(* CODESYS project CowbellCheckers_Tracy.project

Project tree, tasks and I/O mapping:
  Device : PAC320-CXX2X-XX, Parker Hannifin, order no. PAC320-CXX2X-XX, version 3.5.9.10
    application Application
      task EtherCAT_Master (externalevent, external event EVENT_ECM_DC, priority 0) calls EtherCAT_Master.EtherCAT_Task [EtherCAT_Master.EtherCAT_Task], MainProgram
      task VISU_TASK (cyclic, interval 100 ms, priority 31) calls VisuElems.Visu_Prg
      SymbolConfiguration
    SoftMotion General Axis Pool
    EtherCAT_Master : PAC320 EtherCAT Master, Parker Hannifin, order no. PAC320-XXXXX-XX, version 3.5.9.10
      PAC320_BusCoupler : PAC320 BusCoupler, Parker Hannifin, version Revision=16#00000001
          settings: StationAlias = 0; DC sync0 cycletime = 4000; DC sync1 cycletime = 4000
        PACIO_DI16_DO16 : DI16/DO16 1ms 0.5A (PACIO-450-03), Parker Hannifin, version Revision=16#00000001
            settings: StationAlias = 0; DC sync0 cycletime = 4000; DC sync1 cycletime = 4000
            unmapped channels: DigitalOutput0, DigitalOutput1, DigitalOutput2, DigitalOutput3, DigitalOutput4, DigitalOutput5, DigitalOutput6, DigitalOutput7, DigitalOutput8, DigitalOutput9, DigitalOutput10, DigitalOutput11, DigitalOutput12, DigitalOutput13, DigitalOutput14, DigitalOutput15, DigitalInput0, DigitalInput1, DigitalInput2, DigitalInput3, DigitalInput4, DigitalInput5, DigitalInput6, DigitalInput7, DigitalInput8, DigitalInput9, DigitalInput10, DigitalInput11, DigitalInput12, DigitalInput13, DigitalInput14, DigitalInput15
      PD_xxC_Standard_EtherCAT_drive : PD-xxC - Standard EtherCAT drive(CoE,EoE,FoE) V2.0, Parker Hannifin, version Revision=16#00000002
          settings: DC sync0 cycletime = 4000
          unmapped channels: Controlword, Target Position, Touch Probe Function, Digital Ouputs, Statusword, Position Actual Value, Following Error Actual Value, Touch Probe Status, Touch Probe 1 Positive Edge Position Value, Digital Inputs
        X : SM_Drive_GenericDSP402, 3S - Smart Software Solutions GmbH, order no. 0, version 4.0.0.0
            settings: wDriveID = 3; AdrOffset_8010 = 4; BitOffset_8010 = 0; BitLength_8010 = 16; Address_8010 = '%QW2'; Type_8010 = 'UINT'; AddressPointer_8010 = ADR(%QW2); AdrOffset_8020 = 8; BitOffset_8020 = 0; BitLength_8020 = 32; Address_8020 = '%QD2'; Type_8020 = 'DINT'; AddressPointer_8020 = ADR(%QD2); AdrOffset_8030 = 4294967295; BitOffset_8030 = 0; BitLength_8030 = 0; Address_8030 = ''; Type_8030 = ''; AddressPointer_8030 = 0; AdrOffset_8040 = 4294967295; BitOffset_8040 = 0; BitLength_8040 = 0; Address_8040 = ''; Type_8040 = ''; AddressPointer_8040 = 0; AdrOffset_8050 = 4294967295; BitOffset_8050 = 0; BitLength_8050 = 0; Address_8050 = ''; Type_8050 = ''; AddressPointer_8050 = 0; AdrOffset_8060 = 12; BitOffset_8060 = 0; BitLength_8060 = 16; Address_8060 = '%QW6'; Type_8060 = 'UINT'; AddressPointer_8060 = ADR(%QW6); AdrOffset_8070 = 4294967295; BitOffset_8070 = 0; BitLength_8070 = 0;
              Address_8070 = ''; Type_8070 = ''; AddressPointer_8070 = 0; AdrOffset_8080 = 4294967295; BitOffset_8080 = 0; BitLength_8080 = 0; Address_8080 = ''; Type_8080 = ''; AddressPointer_8080 = 0; AdrOffset_8090 = 16; BitOffset_8090 = 0; BitLength_8090 = 32; Address_8090 = '%QD4'; Type_8090 = 'UDINT'; AddressPointer_8090 = ADR(%QD4); AdrOffset_8510 = 4; BitOffset_8510 = 0; BitLength_8510 = 16; Address_8510 = '%IW2'; Type_8510 = 'UINT'; AddressPointer_8510 = ADR(%IW2); AdrOffset_8520 = 8; BitOffset_8520 = 0; BitLength_8520 = 32; Address_8520 = '%ID2'; Type_8520 = 'DINT'; AddressPointer_8520 = ADR(%ID2); AdrOffset_8530 = 4294967295; BitOffset_8530 = 0; BitLength_8530 = 0; Address_8530 = ''; Type_8530 = ''; AddressPointer_8530 = 0; AdrOffset_8540 = 4294967295; BitOffset_8540 = 0; BitLength_8540 = 0; Address_8540 = ''; Type_8540 = ''; AddressPointer_8540 = 0; AdrOffset_8550 = 4294967295;
              BitOffset_8550 = 0; BitLength_8550 = 0; Address_8550 = ''; Type_8550 = ''; AddressPointer_8550 = 0; AdrOffset_8560 = 24; BitOffset_8560 = 0; BitLength_8560 = 32; Address_8560 = '%ID6'; Type_8560 = 'UDINT'; AddressPointer_8560 = ADR(%ID6); AdrOffset_8570 = 16; BitOffset_8570 = 0; BitLength_8570 = 16; Address_8570 = '%IW8'; Type_8570 = 'UINT'; AddressPointer_8570 = ADR(%IW8); AdrOffset_8580 = 20; BitOffset_8580 = 0; BitLength_8580 = 32; Address_8580 = '%ID5'; Type_8580 = 'DINT'; AddressPointer_8580 = ADR(%ID5); AdrOffset_8590 = 4294967295; BitOffset_8590 = 0; BitLength_8590 = 0; Address_8590 = ''; Type_8590 = ''; AddressPointer_8590 = 0; AdrOffset_8600 = 4294967295; BitOffset_8600 = 0; BitLength_8600 = 0; Address_8600 = ''; Type_8600 = ''; AddressPointer_8600 = 0; AdrOffset_8600 = 4294967295; BitOffset_8600 = 0; BitLength_8600 = 0; Address_8610 = ''; Type_8610 = '';
              AddressPointer_8610 = 0; AdrOffset_8620 = 12; BitOffset_8620 = 0; BitLength_8620 = 32; Address_8620 = '%ID3'; Type_8620 = 'DINT'; AddressPointer_8620 = ADR(%ID3)
  CODESYS_SoftMotion_Win_V3 : CODESYS SoftMotion Win V3, 3S - Smart Software Solutions GmbH, order no. 309021, version 3.5.9.10
    application Application
      libraries: PAC Help Library, 0.1 (Parker ); SysFile, 3.5.9.0 (System); CmpErrors, 3.3.1.40 (System); ISysTypes2, 3.5.0.0 (System); SysTimeRtc, 3.5.5.0 (System); SysTimeCore, 3.5.5.0 (System); Util, 3.5.9.0 (System)
      task Main (cyclic, interval 4000 ms, priority 0) calls TestInitialization, TestMyArray
      task VISU_TASK (cyclic, interval 100 ms, priority 31) calls VisuElems.Visu_Prg
      SymbolConfiguration
      Visualizations/
        visualisation Enable
        visualisation OnePlayer
        visualisation InitScreen
        visualisation MainView
        visualisation GameView
        visualisation HowToPlay
        visualisation History
      program TestMyArray [ST]
      global variables PersistentVars
      data type History
      function block ArrayMove [ST]
      program LogData [ST]
      function GetHeaderString [ST]
      function GetTimeStampString [ST]
      program LogWinnerNames [ST]
      function GetLogMsgString [ST]
      visualisation ExportData
    SoftMotion General Axis Pool
      X : SM_Drive_Virtual, 3S - Smart Software Solutions GmbH, order no. 1805, version 4.0.0.0
          settings: wDriveID = 4
      Y : SM_Drive_Virtual, 3S - Smart Software Solutions GmbH, order no. 1805, version 4.0.0.0
          settings: wDriveID = 5
      Z : SM_Drive_Virtual, 3S - Smart Software Solutions GmbH, order no. 1805, version 4.0.0.0
          settings: wDriveID = 6
  text COWBELL_PROGRAMMING_STANDARD
  global variables GlobalVars
  text list GlobalTextList
  function block Initialization [CFC]
  program TestInitialization [CFC]
*)

// CODESYS_SoftMotion_Win_V3/Application/History
TYPE History :
STRUCT
	
	Names: STRING;
	Moves: INT;
	
END_STRUCT
END_TYPE

// GlobalVars
(* COWBELL GLOBAL VARIABLES *)
VAR_GLOBAL
	systemEnable : BOOL;
	
	
	p1CheckerColor: DWORD := 16#FFFFFFFF; // 16# - interpret as hexidecimal, FF - transparency (Fully Opaque, 00 fully transparent), FF - Red, FF - Green, FF - Blue
	p2CheckerColor: DWORD := 16#FF000000;
	
	p1DefaultName: STRING := 'Player_1';
	p2DefaultName: STRING := 'Player_2';
	
	winnerName: STRING := 'Default';
	winnerMoves: INT := 4;
	
	//Export data global variables
	
	g_PosDistance:REAL := 20.0;
	g_NegDistance:REAL := -20.0;
	g_Vel:REAL := 5.0;
	g_Acc:REAL := 10.0;
	//In_Power : BOOL ;
	//In_Reset : BOOL;
	//In_Pos : BOOL;
	//In_Neg : BOOL;
	//In_Stop : BOOL;
	//In_Zero : BOOL;
	g_MoveDwellPos : BOOL := FALSE;
	g_MoveDwellNeg : BOOL := FALSE;
	g_MoveDwellPos_Y : BOOL := FALSE;
	g_MoveDwellNeg_Y : BOOL := FALSE;
	g_MoveDwellPos_Z : BOOL := FALSE;
	g_MoveDwellNeg_Z : BOOL := FALSE;
	g_MoveDwellPos_A : BOOL := FALSE;
	g_MoveDwellNeg_A : BOOL := FALSE;
	g_GotSDO_PostionPos : BOOL;
	g_GotSDO_PostionNeg : BOOL;
	g_GotSDO_Y_PostionPos : BOOL;
	g_GotSDO_Y_PostionNeg : BOOL;
	DC_InSync: BOOL;
	g_FirstSync: BOOL;
	g_LostSync: BOOL;
	
	
	//ScanTimeMax: DINT;
	//ScanTimeMin: DINT;
	//dcWindow: WORD := 50;

	//MaxScanTime: DINT;
	//MaxSyncTime: DINT;
	//MinSyncTime: DINT;
	//MaxTotalSyncBufferAvg: DINT;
	MyArray: ARRAY[0..9, 0..9] OF REAL;
	
END_VAR

// CODESYS_SoftMotion_Win_V3/Application/PersistentVars
{attribute 'qualified_only'}
VAR_GLOBAL PERSISTENT RETAIN
	MyArray : ARRAY [1..20] OF History;
END_VAR

// TestInitialization
PROGRAM TestInitialization
VAR
	Initialization_0: Initialization;
	X_enable: BOOL;
	X_reset: BOOL;
	
END_VAR

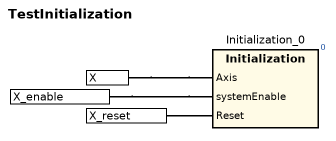
Initialization_0(Axis := X, systemEnable := X_enable, Reset := X_reset); // Initialization

END_PROGRAM

// Initialization
FUNCTION_BLOCK Initialization
VAR_IN_OUT
	Axis: SM3_Basic.AXIS_REF_SM3;
	END_VAR
VAR_INPUT
	systemEnable : BOOL;
	Reset:BOOL;     // reset the drive
	
	
END_VAR
VAR_OUTPUT
END_VAR
VAR
	MC_Power_X: MC_Power;
	MC_Power_Y: MC_Power;
	MC_Power_Z: MC_Power;
	MC_Reset_X: MC_Reset;
	MC_Reset_Y: MC_Reset;
	MC_Reset_Z: MC_Reset;
	MC_Jog_X: MC_Jog;
END_VAR

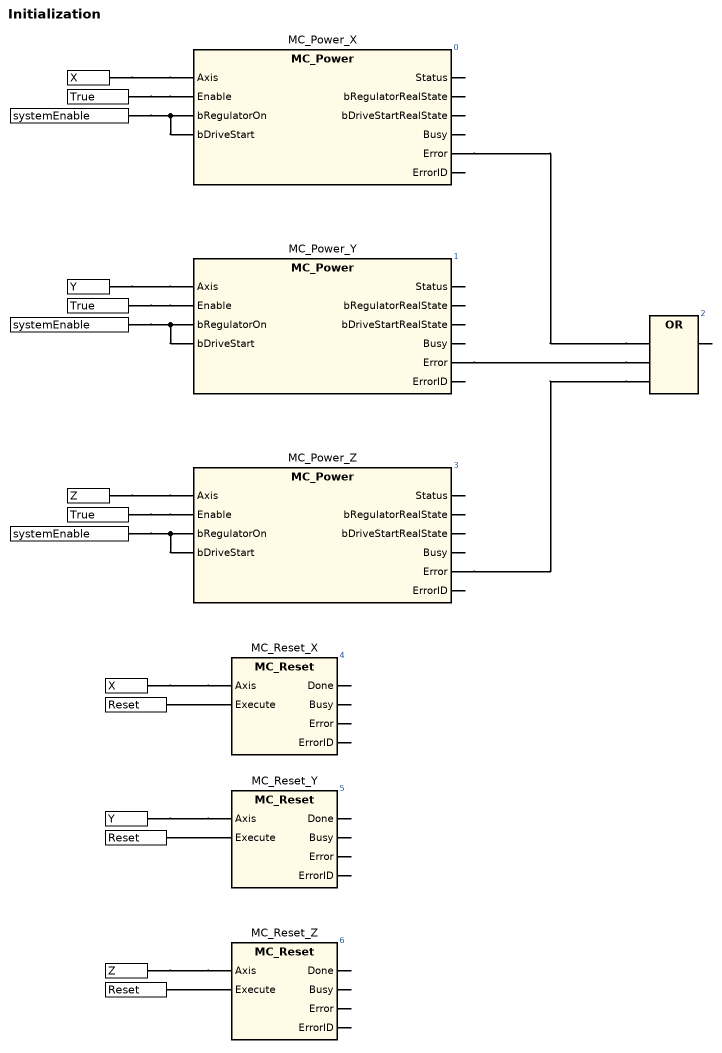
MC_Power_X(Axis := X, Enable := True, bRegulatorOn := systemEnable, bDriveStart := systemEnable); // MC_Power
MC_Power_Y(Axis := Y, Enable := True, bRegulatorOn := systemEnable, bDriveStart := systemEnable); // MC_Power
(* MC_Power_X.Error OR MC_Power_Y.Error OR MC_Power_Z.Error; result not used *)
MC_Power_Z(Axis := Z, Enable := True, bRegulatorOn := systemEnable, bDriveStart := systemEnable); // MC_Power
MC_Reset_X(Axis := X, Execute := Reset); // MC_Reset
MC_Reset_Y(Axis := Y, Execute := Reset); // MC_Reset
MC_Reset_Z(Axis := Z, Execute := Reset); // MC_Reset

END_FUNCTION_BLOCK

// CODESYS_SoftMotion_Win_V3/Application/TestMyArray
PROGRAM TestMyArray
VAR
	k : INT ; 
	arrayTest : ArrayMove;
END_VAR

arrayTest();
//k := ArrayMove.TestArray[2];

END_PROGRAM

// CODESYS_SoftMotion_Win_V3/Application/ArrayMove
FUNCTION_BLOCK ArrayMove
VAR_INPUT
	//TestArray: ARRAY [1..20] OF INT := [1,2,3,4,5,6,7,8,9,10,11,12,13,14,15,16,17,18,19,20];
	i: INT ; 
END_VAR
VAR_OUTPUT
END_VAR
VAR
	Done : BOOL;
END_VAR

IF(NOT Done) THEN
	
FOR i:= 20 TO 2 BY -1 DO 
	PersistentVars.MyArray[i]:= PersistentVars.MyArray [i-1];
END_FOR
PersistentVars.MyArray[1].Names := winnerName;
PersistentVars.MyArray[1].Moves := winnerMoves;
Done := TRUE;
END_IF

END_FUNCTION_BLOCK

// CODESYS_SoftMotion_Win_V3/Application/LogData
PROGRAM LogData
VAR
	filename: STRING := '/Windows/Logs/Log_HighCycleCount.csv';
	filehandle: SYSFILE.RTS_IEC_HANDLE;
	strMsg: STRING[255];
	FOResult: SYSFILE.RTS_IEC_RESULT;
	FWResult: SYSFILE.RTS_IEC_RESULT;
	FWStatus: POINTER TO RTS_IEC_RESULT;
	FCResult: SYSFILE.RTS_IEC_RESULT;
	bytesWritten: DWORD;
	bFileOpen: BOOL;
	iStatus : INT := 0;
	
	
	SafeToStop: BOOL;
	Result1: SYSFILE.RTS_IEC_RESULT;
	SizeFile: DWORD;
	ErrorID: INT;
	diActPosition: UDINT;
	
	LogIndex :DINT := 0;
	LogMsg : ARRAY [1..200] OF STRING[255];
	LogType : STRING;

	intIndex: DINT;
	

END_VAR

CASE iStatus OF
	1: //Open File
	
	SafeToStop := FALSE;
	filehandle := SysFileOpen(szFile := filename, am := sysfile.AM_WRITE, pResult:= ADR(FOResult));
	IF (filehandle <> 16#00000000 AND filehandle <> 16#FFFFFFFF AND FOResult = cmperrors.Errors.ERR_OK) THEN 
		bFileOpen := TRUE;
		iStatus := iStatus + 1;
	ELSE
		ErrorID := -1 * iStatus;  //Open Memory Copy Failed
		iStatus := 99;
	END_IF//Open File

2:	//Log Data
	FOR intIndex := 1 TO LogIndex DO
		strMsg := LogMsg[intIndex];
		bytesWritten:= SysFileWrite(filehandle, ADR(strMsg), DINT_TO_DWORD(LEN(strMsg)), ADR(FWResult));
		IF FWResult <> CmpErrors.Errors.ERR_OK THEN
			ErrorID := -1 * iStatus;  //Log Data Failed
			iStatus := 100;
		END_IF
	END_FOR

3:  //Close File
	FCResult := SysFileClose(filehandle);
	IF FCResult = CmpErrors.Errors.ERR_OK THEN
		SafeToStop:=TRUE;
		iStatus := 5;
	ELSE
		ErrorID := -1 * iStatus;  //File Close Failed
		iStatus := 99;
	END_IF
END_CASE

END_PROGRAM

// CODESYS_SoftMotion_Win_V3/Application/GetHeaderString
FUNCTION GetHeaderString : STRING[255]
VAR_INPUT
END_VAR
VAR
	msg: STRING[255];
	seperator: STRING;
	eol:String;
	strTemp0 : STRING[255];
	strTemp1 : STRING[255];
	

END_VAR

eol := WORD_AS_STRING(16#0A0D, FALSE);
seperator := ',';

strTemp0 := Concat(Concat(	'Winners', 
						 seperator), 
						    'Moves');




GetHeaderString := Concat(Concat(Concat(Concat(	'TimeStamp', 
														seperator),
														strTemp0), 
														seperator),
						     								eol);

END_FUNCTION

// CODESYS_SoftMotion_Win_V3/Application/GetTimeStampString
FUNCTION GetTimeStampString : STRING
VAR_INPUT
END_VAR
VAR
	TimeStamp : SysTime;
	StructTimeStamp : SysTimeDate;
	Result : RTS_IEC_RESULT;
	StrDate : STRING;
	StrTime : STRING;
	

END_VAR

Result := systimertc.SysTimeRtcHighResGet(pTimestamp := TimeStamp);

Result := systimertc.SysTimeRtcConvertHighResToLocal(pTimeStamp:=TimeStamp, pDate:=StructTimeStamp);

StrDate := UINT_TO_STRING(StructTimeStamp.wYear);
IF StructTimeStamp.wMonth < 10 THEN 
	StrDate := Concat(Concat(StrDate, '0') , UINT_TO_STRING(StructTimeStamp.wMonth));
ELSE
	StrDate := Concat(StrDate , UINT_TO_STRING(StructTimeStamp.wMonth));
END_IF

IF StructTimeStamp.wDay < 10 THEN 
	StrDate := Concat(Concat(StrDate , '0') , UINT_TO_STRING(StructTimeStamp.wDay));
ELSE
	StrDate := Concat(StrDate , UINT_TO_STRING(StructTimeStamp.wDay));
END_IF


IF StructTimeStamp.wHour < 10 THEN 
	StrTime := Concat(Concat('0' , UINT_TO_STRING(StructTimeStamp.wHour)) , ':');
ELSE
	StrTime := Concat(UINT_TO_STRING(StructTimeStamp.wHour) , ':');
END_IF

IF StructTimeStamp.wMinute < 10 THEN 
	StrTime := Concat(Concat(Concat(StrTime , '0') , UINT_TO_STRING(StructTimeStamp.wMinute)), ':');
ELSE
	StrTime := Concat(Concat(StrTime , UINT_TO_STRING(StructTimeStamp.wMinute)), ':');
END_IF

IF StructTimeStamp.wSecond < 10 THEN 
	StrTime := Concat(Concat(Concat(StrTime , '0') , UINT_TO_STRING(StructTimeStamp.wSecond)) , '.');
ELSE
	StrTime := Concat(Concat(StrTime , UINT_TO_STRING(StructTimeStamp.wSecond)) , '.');
END_IF

IF StructTimeStamp.wMilliseconds < 10 THEN 
	StrTime := Concat(Concat(StrTime , '00') , UINT_TO_STRING(StructTimeStamp.wMilliseconds));
ELSE
	IF StructTimeStamp.wMilliseconds < 100 THEN 
		StrTime := Concat(Concat(StrTime , '0') , UINT_TO_STRING(StructTimeStamp.wMilliseconds));
	ELSE
		StrTime := Concat(StrTime , UINT_TO_STRING(StructTimeStamp.wMilliseconds));
	END_IF
END_IF

//GetTimeStampString := Concat(Concat(strDate , '-'), strTime);
GetTimeStampString := strTime;

END_FUNCTION

// CODESYS_SoftMotion_Win_V3/Application/LogWinnerNames
PROGRAM LogWinnerNames
VAR
	strMsg: STRING[255];
	iStatus : INT := 0;
	LogIndex :DINT := 0;
	LogMsg : ARRAY [1..200] OF STRING[255];
	LogType : STRING;
	
	CycleTimeWarning: DWORD := 600;
	TotalSyncBufferAvgWarning: DINT := 125;
	CycleTimeError: DWORD := 900;
	TotalSyncBufferAvgError: DINT := 200;
	
	
	
END_VAR

VAR_INPUT
	bResetArray: BOOL;
END_VAR

IF bResetArray = TRUE THEN
	LogIndex := 0;
END_IF




CASE iStatus OF
	

0:	//Log Data
	LogIndex := LogIndex + 1;
	
	LogMsg[LogIndex] :=  GetLogMsgString();
	
	iStatus := 2;

END_CASE

END_PROGRAM

// CODESYS_SoftMotion_Win_V3/Application/GetLogMsgString
FUNCTION GetLogMsgString : STRING[255]
VAR_INPUT
END_VAR
VAR
	msg: STRING[255];
	seperator: STRING;
	eol:String;
	
	DataPrep: STRING[255];
	
	
END_VAR

eol := WORD_AS_STRING(16#0A0D, FALSE);
seperator := ',';


DataPrep := Concat(Concat(  PersistentVars.MyArray[1].Names,
                                                  seperator),
            INT_TO_STRING(PersistentVars.MyArray[1].Moves));
																												



GetLogMsgString := Concat(Concat(Concat(Concat(	GetTimeStampString(),
														seperator),
														DataPrep), 
														seperator),
															eol);

END_FUNCTION

// CODESYS_SoftMotion_Win_V3/Application/Visualizations/Enable
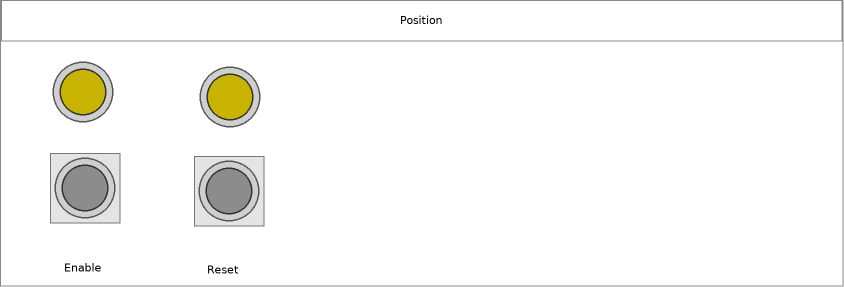
VISUALIZATION Enable  // 844x287
    Frame (1,0 841x41), "Position", text variable: X
        shows SM3_Basic.LinDrive(m_Input_AXISREF := X)
    Label (8,253 150x30), "Enable"
    PushSwitch (50,153 70x70), variable: TestInitialization.X_enable, behaviour: TOGGLE, style: Switch-PushSwitch-Gray
    Lamp1 (48,57 70x70), variable: TestInitialization.X_enable, style: Lamp-Lamp1-Yellow
    PushSwitch (194,156 70x70), variable: TestInitialization.X_reset, behaviour: TOGGLE, style: Switch-PushSwitch-Gray
    Lamp1 (195,62 70x70), variable: TestInitialization.X_reset, style: Lamp-Lamp1-Yellow
    Label (148,255 150x30), "Reset"
END_VISUALIZATION

// CODESYS_SoftMotion_Win_V3/Application/Visualizations/OnePlayer
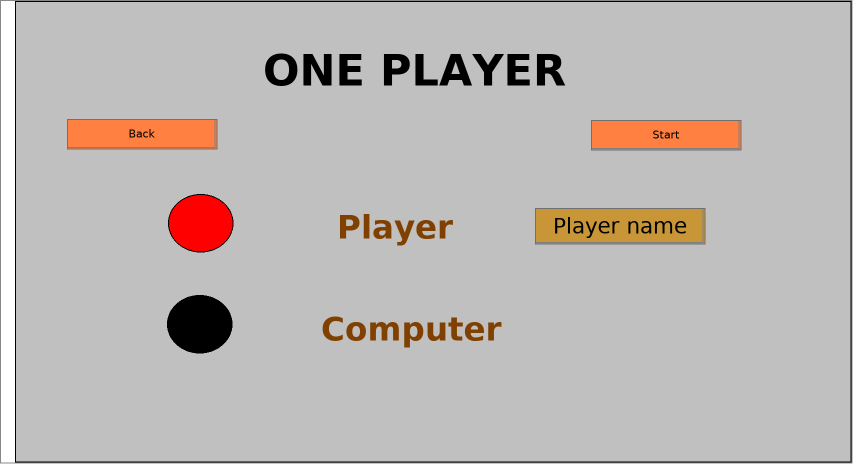
VISUALIZATION OnePlayer  // 853x464
    Rectangle (15,1 836x461)
    Label (230,22 369x97), "ONE PLAYER"
    Button (67,119 150x30), "Back"
    Button (591,120 150x30), "Start"
    Label (326,203 138x48), "Player"
    Button (535,208 170x36), "Player name"
    Ellipse (168,194 65x58)
    Ellipse (167,295 65x58)
    Label (281,305 261x48), "Computer"
END_VISUALIZATION

// CODESYS_SoftMotion_Win_V3/Application/Visualizations/InitScreen
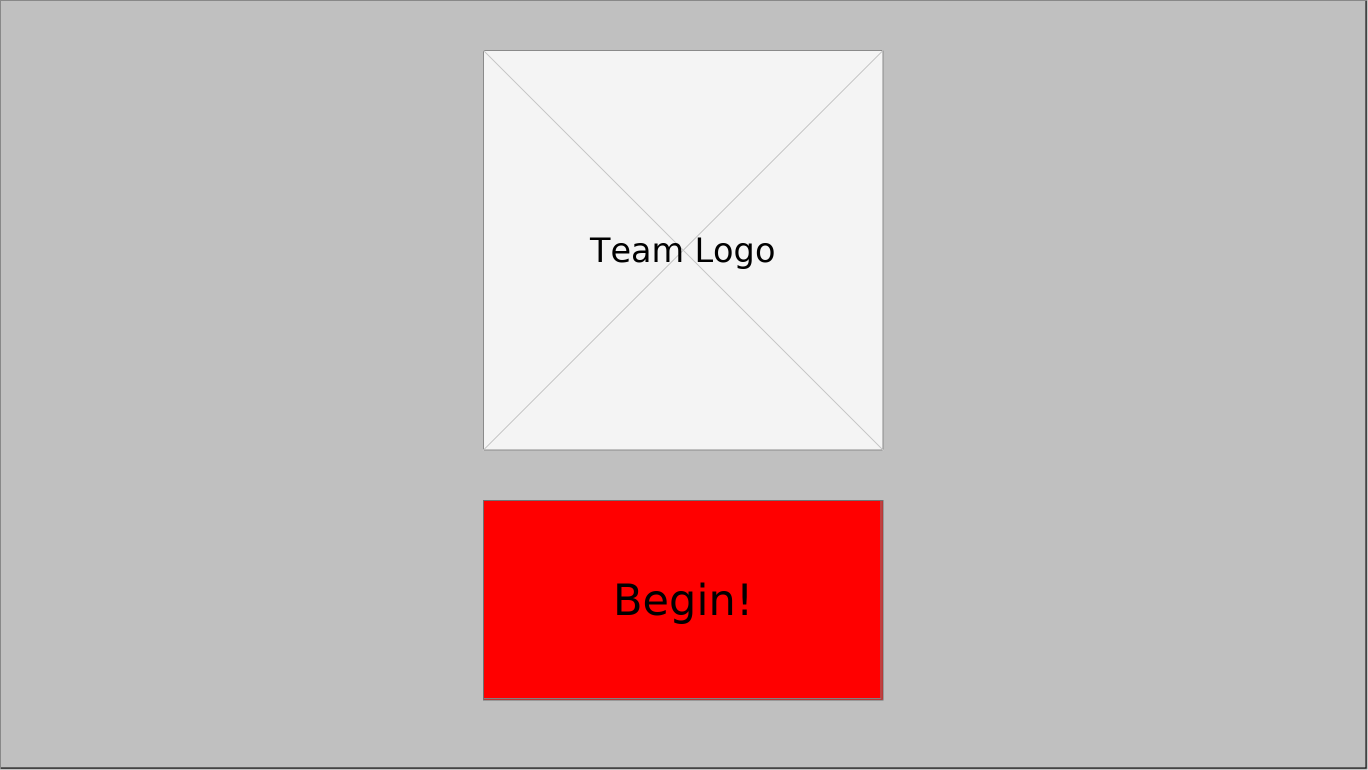
VISUALIZATION InitScreen  // 1368x770
    Rectangle (0,0 1366x768)
    Image (483,50 400x400), "Team Logo"
    Button (483,500 400x200), "Begin!"
END_VISUALIZATION

// CODESYS_SoftMotion_Win_V3/Application/Visualizations/MainView
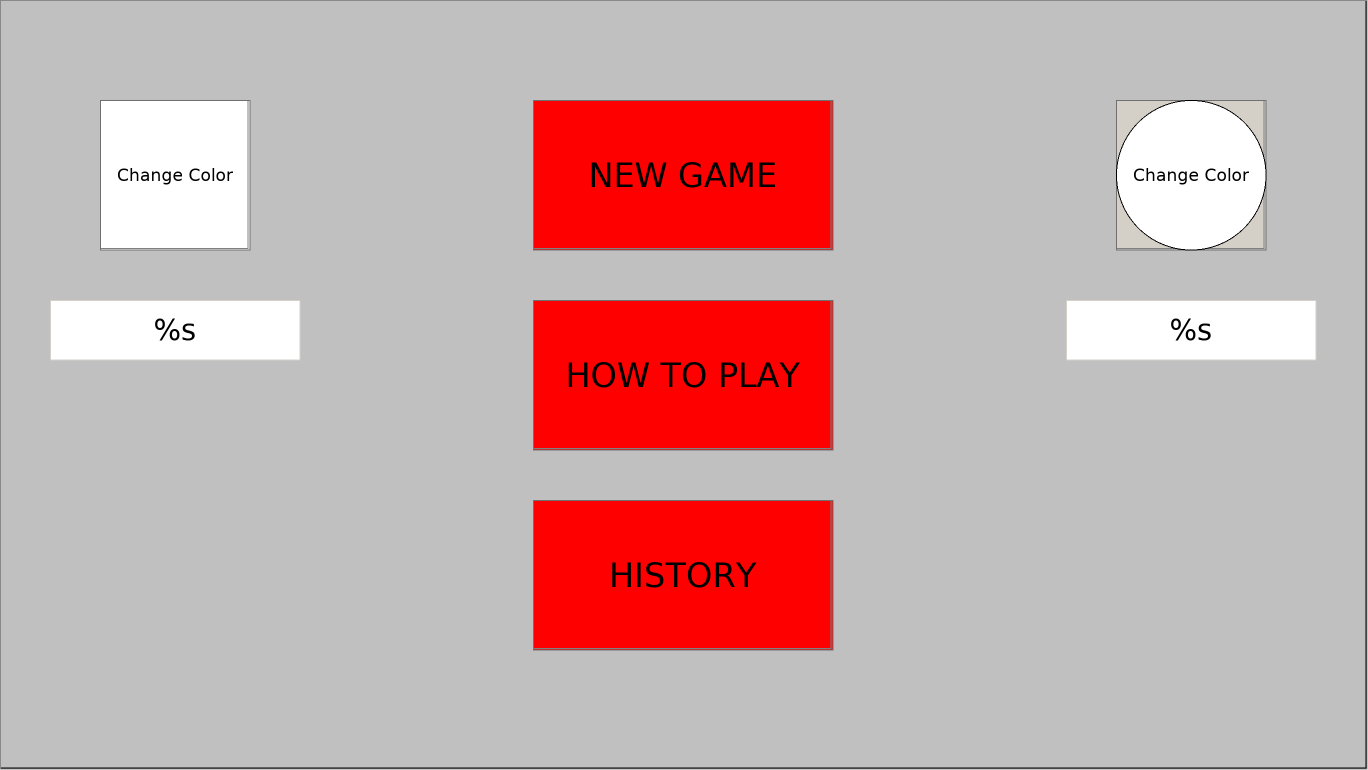
VISUALIZATION MainView  // 1368x770
    Rectangle (0,0 1366x768)
    Ellipse (100,100 150x150), colour variable: p1CheckerColor
    Button (100,100 150x150), "Change Color"
    Button (1116,100 150x150)
    Ellipse (1116,100 150x150), "Change Color", colour variable: p2CheckerColor
    Textfield (50,300 250x60), "%s", text variable: p1DefaultName
    Textfield (1066,300 250x60), "%s", text variable: p2DefaultName
    Button (533,100 300x150), "NEW GAME"
    Button (533,300 300x150), "HOW TO PLAY"
    Button (533,500 300x150), "HISTORY"
END_VISUALIZATION

// CODESYS_SoftMotion_Win_V3/Application/Visualizations/GameView
VISUALIZATION GameView  // 2x2
END_VISUALIZATION

// CODESYS_SoftMotion_Win_V3/Application/Visualizations/HowToPlay
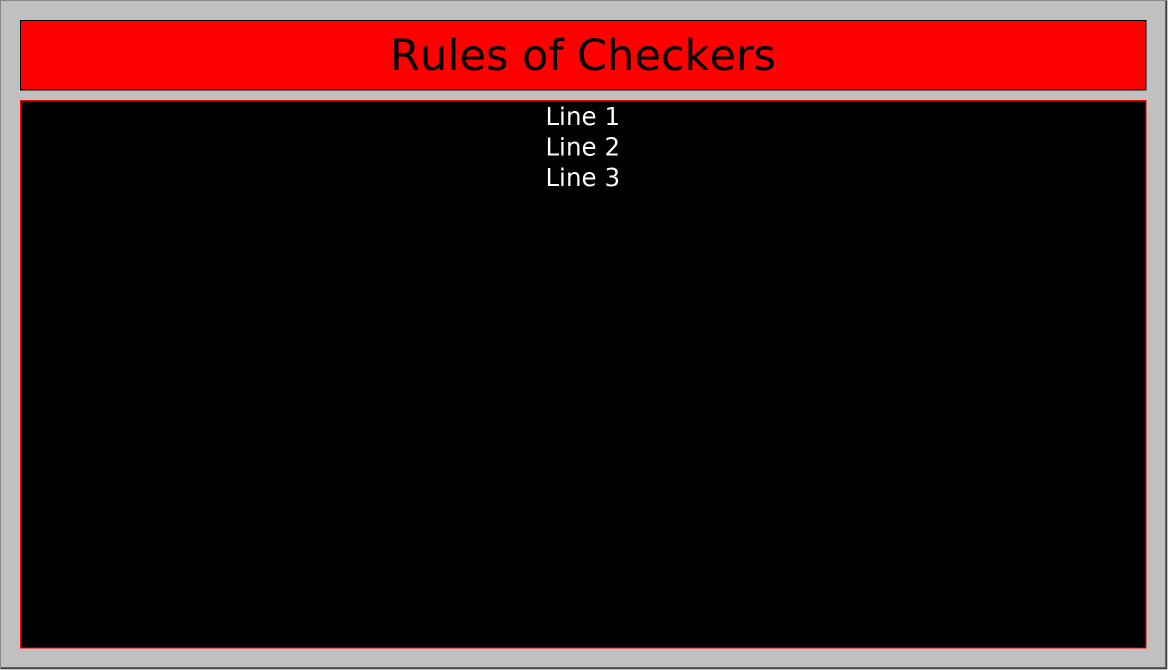
VISUALIZATION HowToPlay  // 1168x670
    Rectangle (0,0 1166x668)
    Textfield (20,100 1126x548), "Line 1 Line 2 Line 3"
    Textfield (20,20 1126x70), "Rules of Checkers"
END_VISUALIZATION

// CODESYS_SoftMotion_Win_V3/Application/Visualizations/History
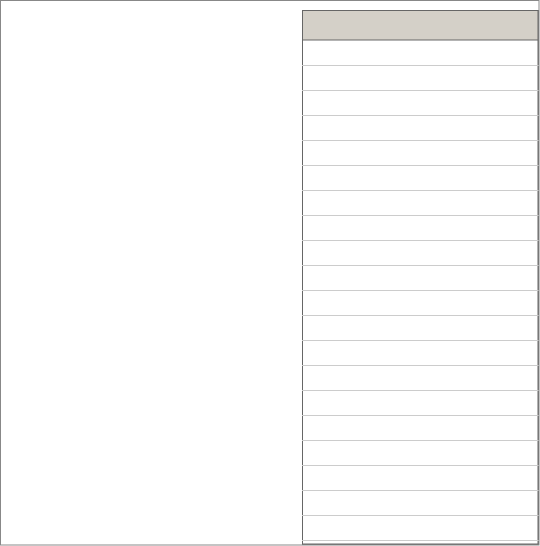
VISUALIZATION History  // 540x546
    Table (302,10 236x534), data array: PersistentVars.MyArray
        p3854506369: PersistentVars.MyArray[INDEX].Names
        p1892666644: PersistentVars.MyArray[INDEX].Moves
        p2232123230: Winners
END_VISUALIZATION

// CODESYS_SoftMotion_Win_V3/Application/ExportData
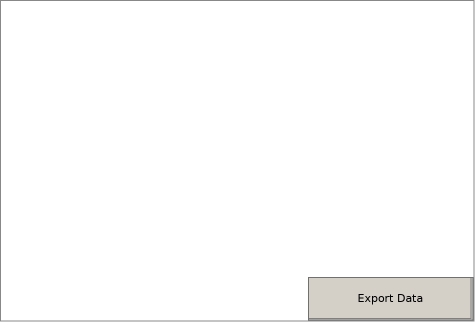
VISUALIZATION ExportData  // 475x322
    Button (308,277 165x43), "Export Data"
END_VISUALIZATION

(* text COWBELL_PROGRAMMING_STANDARD
*** General Team Guidelines ***

Program Names (Func, FB, Prog): ProgramName, Program_Name
-Which ever way appears more readable

Variable Names: var1, xVelocity, yVel1
-If global axis variable, axis identifier leads descriptive name.  start lowercase, camelCase

Functions, FunctionBlocks: These should not use global variables, if it can be avoided.  
These types should be able to copy and paste into a new program.

( * Header Comment * ) - good for describing chuncks of code
// In line comment - good for describing a single line

Programs, GlobalVars, etc. will be placed in the POUs so that we can work with the simulator from home.  Don't forget to copy programs to the required task!


Functions can only be called, take inputs and have defined outputs.  Good for math or modifiers.
Function Blocks must be called in a program and do not have explicitly defined inputs and outputs.  Good for repetive chunks of code.  
Programs are the only items that are run in the Task Configuration list.  Programs will call Functions and Function Blocks as required.  

*For Visual Stuff, let's try to stay with the Arial family of Fonts
*)
